{attribute addProperty BoxType "EL9930-0000-0017"}
{attribute addProperty Id "A_0004_EL9930_0001_0017EL9930_56E76016182.25"}
{attribute addProperty CRC "626071991"}
{attribute addProperty SizeInBites "18"}
{attribute addProperty SizeInBytes "2.25"}
TYPE A_0003_EL9930_0000_0017_255119B7 EXTENDS EL9930_546406CD :
STRUCT
	{attribute addProperty Name "A_0004_EL9930_0001_0017"}
	A_0004_EL9930_0001_0017 : EL9930_56E76016;
END_STRUCT
END_TYPE

(* stored: Version 1.2.0.0, ProductVersion 3.1.4024.9
   DUT A_0003_EL9930_0000_0017_255119B7: Id {1eaa7386-9b9f-4908-be76-91de3d0d528e} *)
